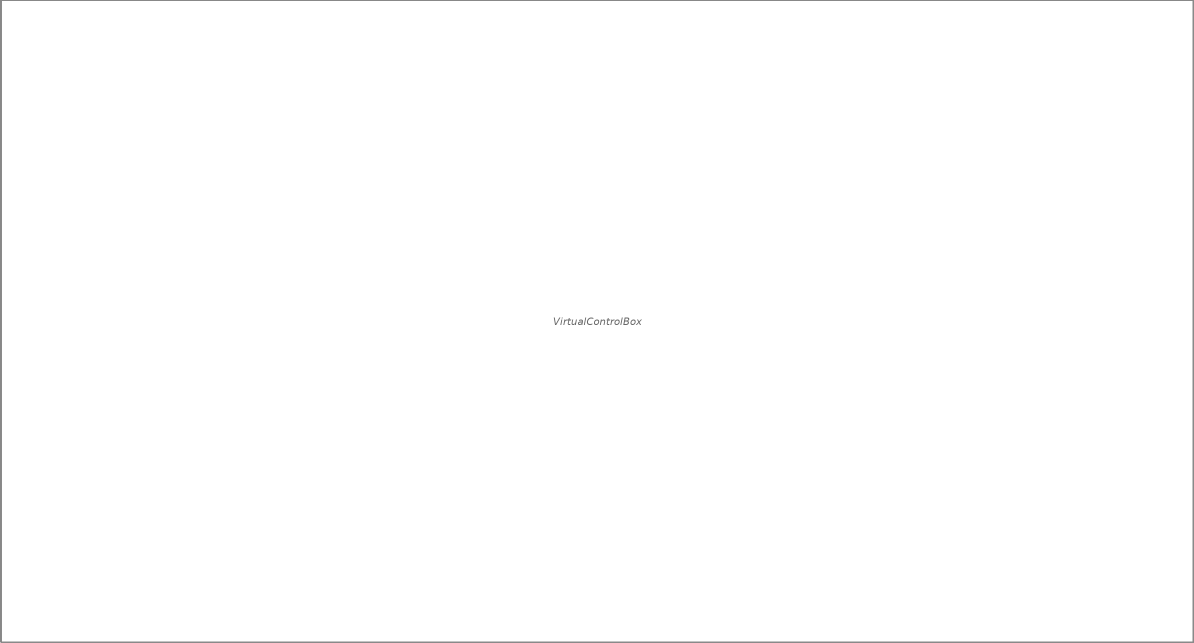
VISUALIZATION HMI  // 1194x643
    TabControl (1,0 1193x643)
        shows VirtualControlBox()
        shows CommissioningHMI()
        shows Animation()
        [0]: TabTitle=ControlBox
        [1]: TabTitle=Comissioning
        [2]: TabTitle=Animation
END_VISUALIZATION

(* stored: Version 1.1.0.1, ProductVersion 3.1.4024.12
   Visu HMI: Id {8f001f6a-c295-4012-bff0-8e8a1e7d1481} *)
